Fanuc KAREL source: kt00098.KL

PROGRAM KT00098
%NOLOCKGROUP
VAR
I1:INTEGER;I2:INTEGER;OUT:REAL
BEGIN
--
--
I1=2
I2=3
I1=2
I2=3
OUT=(I1/(I2))
END KT00098
